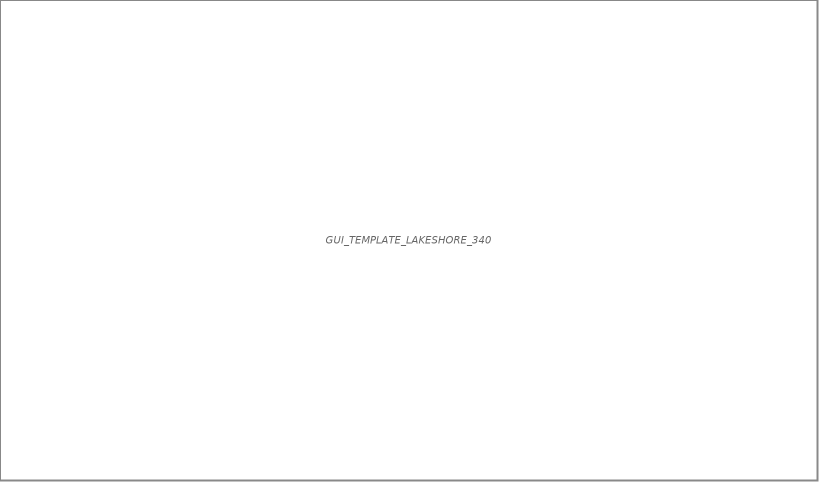
VISUALIZATION GUI_LAKESHORE_340  // 819x482
    Frame (0,0 817x480)
        shows GUI_TEMPLATE_LAKESHORE_340(m_Instance := MAIN.LS340)
END_VISUALIZATION

(* stored: Version 1.1.0.1, ProductVersion 3.1.4022.16
   Visu GUI_LAKESHORE_340: Id {af2819a4-57b0-4877-b8df-4ef57ede2bf3} *)
